FUNCTION_BLOCK HaltMoverTask  IMPLEMENTS I_Task, I_Object, I_Cyclic, I_Abortable
VAR
	haltMoverCA : Tc3_McCollisionAvoidance.MC_HaltCA;
	_Axis : REFERENCE TO Tc2_MC2.AXIS_REF;
	_Error: BOOL;
	_ErrorID: UDINT;
	_Done: BOOL;
END_VAR

{analysis -2}

METHOD Abort : Hresult
haltMoverCA.Execute := FALSE;
END_METHOD

PROPERTY AxisRef : reference to Axis_ref
GET
AxisRef	REF= _Axis;
END_GET
SET
_Axis REF= AxisRef;
END_SET
END_PROPERTY

PROPERTY Busy : BOOL
GET
Busy := haltMoverCA.Busy;
END_GET
END_PROPERTY

METHOD Cycle : HRESULT
VAR_INPUT
END_VAR
IF NOT __ISVALIDREF(_Axis) THEN
	Cycle := -1;
	RETURN;
END_IF

haltMoverCA(Axis := _Axis);
_Done := haltMoverCA.Done OR _Done;
_Error := haltMoverCA.Error OR _Error;
IF haltMoverCA.ErrorId <> 0 THEN
	_ErrorID := haltMoverCA.ErrorId;
END_IF
haltMoverCA.Execute := false;
END_METHOD

PROPERTY Deceleration : MC_LREAL
GET
Deceleration := haltMoverCA.Deceleration;
END_GET
SET
IF Deceleration > 0.0 THEN
	haltMoverCA.Deceleration := Deceleration;
END_IF
END_SET
END_PROPERTY

PROPERTY Done : BOOL
GET
Done := _Done;
END_GET
END_PROPERTY

PROPERTY Error : BOOL
GET
Error := _Error;
END_GET
END_PROPERTY

METHOD Execute : HRESULT
VAR_INPUT
END_VAR
IF haltMoverCA.Execute THEN
	Execute := -1;
	RETURN;
END_IF

IF NOT __ISVALIDREF(_axis) THEN
	Execute	 := -1;
	RETURN;
END_IF

haltMoverCA.Execute := TRUE;
_Error := FALSE;
_ErrorId := 0;
_Done := FALSE;
END_METHOD

PROPERTY Gap : MC_LREAL
GET
Gap := haltMoverCA.Gap;
END_GET
SET
IF Gap > 50.0 THEN
	haltMoverCA.Gap := Gap;
END_IF
END_SET
END_PROPERTY

PROPERTY Jerk : MC_LREAL
GET
Jerk := haltMoverCA.Jerk;
END_GET
SET
IF Jerk > 0.0 THEN
	haltMoverCA.Jerk := Jerk;
END_IF
END_SET
END_PROPERTY

METHOD RegisterWithParent
VAR_INPUT
	Parent	: Base_Library.I_HostObjects;
END_VAR
Parent.RegisterCyclic(THIS^);
Parent.RegisterAbortable(THIS^);
Parent.RegisterTask(THIS^);
END_METHOD

END_FUNCTION_BLOCK

(* stored: Version 1.1.0.1
   POU HaltMoverTask: Id {16fe934f-2b92-45c5-becd-cbf7a242dbb1}, SpecialFunc None
   Method Abort: Id {48a4c415-0254-4332-8d1a-2734e5dda505}
   Property AxisRef: Id {a9bddd31-e205-4bbe-b0be-0bb7ddf7f5e3}
   Get Get: Id {0e3b6af2-4e89-4c29-9315-30e22f8c6b94}
   Set Set: Id {0e14ea90-18e4-4a1c-9f4c-2cea8c3719c9}
   Property Busy: Id {410b2236-4b2d-41d8-b891-c048fa414dcc}
   Get Get: Id {5856c273-62b7-4af7-b86e-de01e6cc2e07}
   Method Cycle: Id {1e7367c4-25b5-40fa-b219-770d9b7044ce}
   Property Deceleration: Id {c87d7270-1a2e-466f-a142-6139e2eda06f}
   Get Get: Id {a049ca93-b85d-4787-b520-72ad6ac74f0d}
   Set Set: Id {ae2611d3-59b2-4268-a7c2-500b25ff0ec0}
   Property Done: Id {a09eb2b9-def0-4c01-868b-84cd3b62dc56}
   Get Get: Id {a5814443-bbb5-4f85-a263-8110f08b71d3}
   Property Error: Id {6bb2ee39-e78a-4989-a5b3-4f1b4a227870}
   Get Get: Id {206c977d-3fc3-4519-bfba-0ba62f311fe7}
   Method Execute: Id {87eca2aa-365e-4c2f-b198-b62e8029fb82}
   Property Gap: Id {a94177ce-b18c-4479-ae6f-5707566b0317}
   Get Get: Id {ec2ed493-6955-4aef-baef-795d6fef3927}
   Set Set: Id {43b68502-e2f4-4b37-a3be-43a3ab3afcec}
   Property Jerk: Id {36146f01-bab8-49f7-9914-96e1977269b5}
   Get Get: Id {bd60b227-3eb3-44e9-be6f-0a525b541f10}
   Set Set: Id {356145f4-af65-48cf-aa74-d0bf709b5382}
   Method RegisterWithParent: Id {1eb21580-73b7-42fe-bf94-583ead68438b} *)
